ELSE
	sQuery := 'select * from t_log where severity = NULL';
END_IF
IF xFilterByDate THEN
	STU.StrConcatA(pstTo := ADR(sQuery), pstFrom := ADR(' AND timestamp < '), iBufferSize := TO_INT(XSIZEOF(sQuery)));
	SysMem.SysMemSet(pDest := ADR(sAux), udiCount := XSIZEOF(sAux), udiValue := 0);
	sAux := SysD_DB.FUN_ConvertToSQLQueryString(sString := sFilter_LastEventDT);
	STU.StrConcatA(pstTo := ADR(sQuery), pstFrom := ADR(sAux), iBufferSize := TO_INT(XSIZEOF(sQuery)));
END_IF
IF xFilterByComponent THEN
	STU.StrConcatA(pstTo := ADR(sQuery), pstFrom := ADR(' AND component = '), iBufferSize := TO_INT(XSIZEOF(sQuery)));
	SysMem.SysMemSet(pDest := ADR(sAux), udiCount := XSIZEOF(sAux), udiValue := 0);
	sAux := SysD_DB.FUN_ConvertToSQLQueryString(sString := sFilter_Component);
	STU.StrConcatA(pstTo := ADR(sQuery), pstFrom := ADR(sAux), iBufferSize := TO_INT(XSIZEOF(sQuery)));
END_IF

xContinueGetLog := xAppendToExtendedLog AND diLastNonNullLogID > 0;//02/11/2022
IF xContinueGetLog THEN //02/11/2022
	STU.StrConcatA(pstTo := ADR(sQuery), pstFrom := ADR(' AND id < '), iBufferSize := TO_INT(XSIZEOF(sQuery)));
	sAux := TO_STRING(diLastNonNullLogID);
	STU.StrConcatA(pstTo := ADR(sQuery), pstFrom := ADR(sAux), iBufferSize := TO_INT(XSIZEOF(sQuery)));
END_IF

STU.StrConcatA(pstTo := ADR(sQuery), pstFrom := ADR(' order by id desc limit 40'), iBufferSize := TO_INT(XSIZEOF(sQuery)));

diQueryLength := STU.StrLenA(pstData := ADR(sQuery));

eQueryError := SysD_DB.FUN_Query2SQLCmd(
	pbQuery := ADR(sQuery), 
	diQueryLength := diQueryLength,
	asSQLCommand => asMySQLCommand	
);

SysMem.SysMemSet(pDest := ADR(aLog), udiCount := XSIZEOF(aLog), udiValue := 0);

pInterpDest := ADR(aLog);
uiDimInterpDest := __UXINT_TO_UINT(XSIZEOF(aLog)/XSIZEOF(aLog[0]));

itfInterpreter := SQL_Interp_GetLog_0;

REF_REQ_SQLQuery REF= REQ_GetLog;

eMySQLAction := SysD_DB.SysD_DB_actions_enum_t.Query;


                      
END_ACTION

ACTION ACT_GetLog_Success:
                        IF eLastInterpError = SysD_DB.ERROR.NO_ERROR THEN
// 	diActionID := aSAPA_RequestedActions[0].diID;
	METH_CopyToExtendedLog();
ELSIF eLastInterpError = SysD_DB.ERROR.NULL_RESULT THEN
	diActionID := -1;
END_IF
                      
END_ACTION

ACTION ACT_SingleInsert:
                        // SINGLE INSERT
ePollRes := itfQueue_LogEntries.Poll(itfElement => itfElement);
xResult := __QUERYINTERFACE(itfElement, itfLogEntryElement);
IF xResult THEN
	LogEntryToInsert := itfLogEntryElement.LogEntry;
	xLogEntryIsValid := METH_LogEntryIsValid(LogEntry := LogEntryToInsert);
	IF xLogEntryIsValid THEN // single insert
		xTB_InsertLogEntry := TRUE;
	END_IF
END_IF
                      
END_ACTION

ACTION ACT_MultiInsert:
                        ePollRes := COL.COLLECTION_ERROR.NO_ERROR;
sMultiInsertQuery := '';
WHILE METH_MultiInsertCond() DO
	diMultiInsertQueryLen := STU.StrLenA(pstData := ADR(sMultiInsertQuery));
	
	ePeekRes := itfQueue_LogEntries.Peek(itfElement => itfElement);
	xResult := __QUERYINTERFACE(itfElement, itfLogEntryElement);
	IF xResult THEN
		LogEntryToInsert := itfLogEntryElement.LogEntry;
		xLogEntryIsValid := METH_LogEntryIsValid(LogEntry := LogEntryToInsert);
		IF xLogEntryIsValid THEN
			sPeekQuery := '';
			sPeekQuery := FUN_DB_insert_log_entry(
				SysD_LogEntry := LogEntryToInsert,
			);
			
			diPeekQueryLen := STU.StrLenA(pstData := ADR(sPeekQuery));
			diSumQueryLen := diMultiInsertQueryLen + diPeekQueryLen;
			diMaxQueryLen := TO_DINT(XSIZEOF(sMultiInsertQuery)) - 1;
			xAddToMultiInsert := diSumQueryLen < diMaxQueryLen;
			IF xAddToMultiInsert THEN
				// concatenate the peeked string to the query
				xConcatRes := STU.StrConcatA(
					pstTo := ADR(sMultiInsertQuery), 
					pstFrom := ADR(sPeekQuery), 
					iBufferSize := TO_INT(XSIZEOF(sMultiInsertQuery))
				);
				ePollRes := itfQueue_LogEntries.Poll(itfElement => itfElement); // poll the element
			ELSE // don't poll, leave it for the next round
				EXIT;
			END_IF
		ELSE // eliminate by polling
			eRemoveRes := itfQueue_LogEntries.Poll(itfElement => itfElement);
		END_IF
	END_IF
END_WHILE
IF sMultiInsertQuery <> '' THEN
	xTB_MultiInsertLogEntries := TRUE;
END_IF
                      
END_ACTION

METHOD METH_LogEntryIsValid : BOOL
  VAR_INPUT
    LogEntry : SysD_log_entry_t;
  END_VAR
                          METH_LogEntryIsValid := 
	LogEntry.sTimeStamp <> ''
	AND LogEntry.sDescription <> ''
;
                        
END_METHOD

METHOD METH_GetLastNonNullID : DINT
  VAR_INPUT
    pLog : POINTER TO SysD_log_row_t;
    udiDim : UDINT;
  END_VAR
  VAR_OUTPUT
    udiArrayInd : UDINT := 0;
    xEmptyArray : BOOL := TRUE;
  END_VAR
  VAR
    udiInd : UDINT;
    pCurrentLog : POINTER TO SysD_log_row_t;
    diRes : DINT := -1;
    xParsingOK : BOOL;
  END_VAR
                          xParsingOK := pLog > 0 AND udiDim > 0;
IF xParsingOK THEN
	WHILE udiInd < udiDim DO
		pCurrentLog := pLog + TO___XWORD(udiInd) * XSIZEOF(pLog^);
		IF pCurrentLog^.diID = 0 THEN
			EXIT;
		ELSE
			xEmptyArray := FALSE;
			diRes := pCurrentLog^.diID;
			udiArrayInd := udiInd;
			udiInd := udiInd + 1;
		END_IF
	END_WHILE
END_IF

METH_GetLastNonNullID := diRes;
                        
END_METHOD

METHOD METH_CopyToExtendedLog : BOOL
  VAR
    udiExtLastNonNullArrInd : UDINT;
    xExtIsEmptyArray : BOOL;
    diExtLastNonNullLogID : DINT;
    diLocalLastNonNullLogID : DINT;
    xLocalIsEmptyArray : BOOL;
    udiLocalLastNonNullArrInd : UDINT;
    udiExtInd : UDINT;  (* where to copy *)
    udiLocalInd : UDINT;  (* what to copy *)
    pCurrExt : POINTER TO SysD_log_row_t;
    pCurrLocal : POINTER TO SysD_log_row_t;
  END_VAR
                          diExtLastNonNullLogID := METH_GetLastNonNullID(
	pLog := ADR(aExtendedLog), udiDim := udiDimExtendedLog,
	udiArrayInd => udiExtLastNonNullArrInd,
	xEmptyArray => xExtIsEmptyArray
);

diLocalLastNonNullLogID := METH_GetLastNonNullID(
	pLog := ADR(aLog), udiDim := udiDimLog,
	udiArrayInd => udiLocalLastNonNullArrInd,
	xEmptyArray => xLocalIsEmptyArray
);

IF xExtIsEmptyArray THEN
	udiExtInd := 0;
ELSE
	udiExtInd := udiExtLastNonNullArrInd + 1;
END_IF
udiLocalInd := 0;
WHILE udiExtInd < udiDimExtendedLog AND udiLocalInd <= udiLocalLastNonNullArrInd DO
	pCurrExt := ADR(aExtendedLog) + udiExtInd * XSIZEOF(pCurrExt^);
	pCurrLocal := ADR(aLog) + udiLocalInd * XSIZEOF(pCurrExt^);
	pCurrExt^ := pCurrLocal^; //copy
	
	udiExtInd := udiExtInd + 1;
	udiLocalInd := udiLocalInd + 1;
END_WHILE
                        
END_METHOD

METHOD METH_AddEntryToQueue : COL.COLLECTION_ERROR
  VAR_INPUT
    LogEntry : SysD_log_entry_t;
    pdiCounter : POINTER TO DINT := 0;
  END_VAR
  VAR_OUTPUT
    xFullBuffer : BOOL;
    sLastTimestamp : STRING;
  END_VAR
  VAR
    eRes : COL.COLLECTION_ERROR;
    xAddOk : BOOL;
  END_VAR
                          LogEntry.sTimeStamp := FUN_GetLocalRTCString();
eRes := itfQueue_LogEntries.AddElement(
	itfElement := LogEntriesFactory.Create(
		Value := LogEntry, 
		eError => eLogEntryFactErr
	)
);
xAddOk := eRes = COL.COLLECTION_ERROR.NO_ERROR AND eLogEntryFactErr = FBF.ERROR.NO_ERROR;
IF xAddOk THEN
// 	diCounter := (diCounter + 1) MOD 16#7FFFFFFF;
	IF pdiCounter > 0 THEN //increment counter if passed as pointer
		pdiCounter^ := pdiCounter^ + 1;
	END_IF
	sLastTimestamp := LogEntry.sTimeStamp;
ELSE
	xFullBuffer := eRes = COL.COLLECTION_ERROR.MAXIMUM_SIZE_OF_ELEMENTS_EXCEEDED;
END_IF
                        
END_METHOD

METHOD METH_MultiInsertCond : BOOL
  VAR
    udiEntries : UDINT;
    diMaxQueryLen : DINT;
    diQueryLenThreshold : DINT;
  END_VAR
                          udiEntriesToInsert := itfQueue_LogEntries.CountElements();
diMultiInsertQueryLen := STU.StrLenA(pstData := ADR(sMultiInsertQuery));
diMaxQueryLen := TO_DINT(XSIZEOF(sQuery)) - 1;
diQueryLenThreshold := TO_DINT(TO_REAL(diMaxQueryLen) * 0.75);
// diPeekQueryLen := STU.StrLenA(pstData := ADR(sPeekQuery));

METH_MultiInsertCond :=
	ePollRes = COL.COLLECTION_ERROR.NO_ERROR
	AND udiEntriesToInsert > 0
	AND diMultiInsertQueryLen < diQueryLenThreshold;
;
                        
END_METHOD
END_PROGRAM

PROGRAM prgDBExecutor
  VAR
    eIterResult : COL.COLLECTION_ERROR;
    COL_ListIterator : COL.ListIterator;
    itfStringElement : COL.IElement;
    itfMySQLResult : SysD_DB.IMySQLResultElement;
    xResultIt : BOOL;
    iftStringKey : COL.IStringElement;
    itfElement : COL.IElement;
    xInspectHashtable : BOOL;
    MySQLResult : SysD_DB.SysD_DB_result_struct_t;
    xInspectQueue : BOOL;
    eIterRequest : COL.COLLECTION_ERROR;
    itfMySQLRequest : SysD_DB.IMySQLRequestElement;
    MySQLRequest : SysD_DB.SysD_DB_request_struct_t;
    sTestDBName : STRING := 'db_sapa_test';
    xTB_TESTDB : BOOL;
    xIsTest : BOOL;
    asIN_MySQLRequests : ARRAY[0..c_uiMaxIndArray] OF SysD_DB.IMySQLRequestElement;  (* QUEUE IN *)
    itfINQueue_MySQLRequest : COL.Queue := (paElements := ADR(asIN_MySQLRequests), udiMaxElements := UINT_TO_UDINT((c_uiMaxIndArray + 1)));
    HashTableFactory : COL.HashTableFactory;  (* Factory to create a hash table on heap memory. *)
    itfOUTHashTable_MySQLResult : COL.IMap := HashTableFactory.Create(udiMaxElements := UINT_TO_UDINT((c_uiMaxIndArray + 1)));  (* Creates a hashtable on heap memory. NOTE: Collections that have been created with this Factory are not online change safe. *)
    iCountFailure : INT;
    eLastExecutorError : SysD_DB.EXECUTOR_ERROR;
    udiINRequestsNum : UDINT;
    udiOUTResultsNum : UDINT;
    iMaxClients : INT := 2;
    SysD_DB_Executor_0 : SysD_DB.SysD_DB_Executor;
    CTRL_Executor : SysDesignBasic.SysD_basic_ctrl_struct_t := (xExecute := TRUE);
    eMySQLExecutorError : SysD_DB.EXECUTOR_ERROR;
    ClientsOccupationStatistic : SysD_DB.SysD_DB_clients_occ_stat_struct_t;
    aeClientsOccupation : ARRAY[0..SysD_DB.Constants.gc_uiMaxIndMySQLClients] OF SysD_DB.SysD_DB_client_state_enum_t;
  END_VAR
  VAR CONSTANT
    c_uiMaxIndArray : UINT := 49;
  END_VAR

                    (*--------------------------*)
// 2/12/2022: set database

(*--------------------------*)

udiINRequestsNum := itfINQueue_MySQLRequest.CountElements();
udiOUTResultsNum := itfOUTHashTable_MySQLResult.CountKeys();

SysD_DB_Executor_0(
	xEnable := CTRL_Executor.xExecute,
	xBusy => CTRL_Executor.xProcessing,
	xError => CTRL_Executor.xFailure,
	
	eErrorID => eMySQLExecutorError,
	
	pIN_Queue := ADR(itfINQueue_MySQLRequest),
	pOUT_Hashtable := ADR(itfOUTHashTable_MySQLResult),
	iMaxClients := iMaxClients,
	
	ClientsOccupationStatistic => ClientsOccupationStatistic,
	aeClientsOccupation => aeClientsOccupation
);
CTRL_Executor.xTerminated := CTRL_Executor.xFailure;
IF CTRL_Executor.xTerminated THEN
	eLastExecutorError := eMySQLExecutorError;
	IF CTRL_Executor.xSuccess THEN
		// never
	ELSIF CTRL_Executor.xFailure THEN
		iCountFailure := (iCountFailure + 1) MOD 16#7FFF;
	END_IF
	CTRL_Executor.xExecute := FALSE;
	SysD_DB_Executor_0(xEnable := FALSE);
END_IF
(*=====================================================*)
//21/12/2022: debugging
// IF xInspectHashtable THEN
// 	eIterResult := itfOUTHashTable_MySQLResult.Keys(itfIterator := COL_ListIterator);
// 	IF eIterResult = COL.COLLECTION_ERROR.NO_ERROR THEN
// 		WHILE COL_ListIterator.HasNext() DO
// 			COL_ListIterator.Next(itfElement => itfStringElement);
// 			xResultIt :=  __QUERYINTERFACE(itfStringElement, iftStringKey);
// 			IF xResultIt THEN
// 				itfOUTHashTable_MySQLResult.GetElementByKey(itfKey := iftStringKey, itfValue => itfElement);
// 				xResultIt :=  __QUERYINTERFACE(itfElement, itfMySQLResult);
// 				IF xResultIt THEN 
// 					MySQLResult := itfMySQLResult.PROP_MySQLResultElement;
// 				END_IF
// 			END_IF
// 		END_WHILE;
// 	END_IF
// END_IF
// IF xInspectQueue THEN
// 	eIterRequest := itfINQueue_MySQLRequest.ElementIterator(itfIterator := COL_ListIterator);
// 	IF eIterRequest = COL.COLLECTION_ERROR.NO_ERROR THEN
// 		WHILE COL_ListIterator.HasNext() DO
// 			COL_ListIterator.Next(itfElement => itfElement);
// 			xResultIt :=  __QUERYINTERFACE(itfElement, itfMySQLRequest);
// 			IF xResultIt THEN
// 				MySQLRequest := itfMySQLRequest.PROP_MySQLRequestElement;
// 			END_IF
// 		END_WHILE;
// 	END_IF
// END_IF

                  
END_PROGRAM

(* Implicitly generated code : DO NOT EDIT *)
{attribute 'check_pointer'}
{attribute 'no_check'}
FUNCTION CheckPointer : POINTER TO BYTE
  VAR_INPUT
    ptToTest : POINTER TO BYTE;  (* Destination address of the pointer *)
    iSize : DINT;  (* Size of the type the pointer points to. (e.g: 20 for POINTER TO ARRAY [0..9] OF INT) *)
    iGran : DINT;  (* Granularity of the pointer access. This is the size of the biggest non-structured data type in the type the pointer points to. (e.g: 2 for POINTER TO ARRAY [0..9] OF INT) *)
    bWrite : BOOL;  (* Indicates read or write access. TRUE = write access. *)
  END_VAR
  VAR
    xError : BOOL;
  END_VAR

                    // No standard way of implementation. Fill your own code here.
IF ptToTest = 0 THEN
	xError := TRUE;
END_IF
CheckPointer := ptToTest;
                  
END_FUNCTION

PROGRAM prgInboundSync
  VAR
    BoxAtGateInfo : INCAS_box_info_struct_t;
    xNewBox : BOOL;
    sBoxInfoFromDB : db_t_items_struct_t;
    xInfoReceived : BOOL;
    xDelayBoxInMachineCond : BOOL;
    TON_DelayBoxInMachine : TON;
    tDelay : TIME := TIME#5s0ms;
    BoxAckFeedback : INCAS_box_ack_struct_t;
    iResSetFeedback : INT;
    iAnalyzeRes : INT;
    eErrorID : INCAS_box_error_enum_t;
  END_VAR

                    (*-----------------------------------------*)
// New box on OPC UA
IF xNewBox THEN
	xNewBox := FALSE;
	prgDBQuerier_SorterSX.METH_GetBoxInfo(sBoxCode := BoxAtGateInfo.box_code);
	SysMemSet(pDest := ADR(BoxAckFeedback), udiCount := XSIZEOF(BoxAckFeedback), udiValue := 0);
	BoxAckFeedback.last_box_code := BoxAtGateInfo.box_code;
	BoxAckFeedback.time_stamp := FUN_GetLocalRTCString();
	BoxAckFeedback.error_id := TO_INT(INCAS_box_error_enum_t.BUSY);
	iResSetFeedback := prgOPCUAIncas.METH_SetIncasInboundFeedback_01(
		Feedback := BoxAckFeedback
	);
END_IF
(*-----------------------------------------*)
// info received from DB
IF xInfoReceived THEN
	xInfoReceived := FALSE;
	iAnalyzeRes := METH_AnalyzeBoxInfo(
		InfoOnOPCUa := BoxAtGateInfo,
		InfoOnDb := sBoxInfoFromDB,
		eErrorID => eErrorID
	);
	xDelayBoxInMachineCond := TRUE;
	BoxAckFeedback.time_stamp := FUN_GetLocalRTCString();
	BoxAckFeedback.error_id := TO_INT(eErrorID);
	iResSetFeedback := prgOPCUAIncas.METH_SetIncasInboundFeedback_01(
		Feedback := BoxAckFeedback
	);
END_IF
(*-----------------------------------------*)
// take over
TON_DelayBoxInMachine(IN := xDelayBoxInMachineCond, PT := tDelay);
IF TON_DelayBoxInMachine.Q THEN
	xDelayBoxInMachineCond := FALSE;
	BoxAckFeedback.time_stamp := FUN_GetLocalRTCString();
	BoxAckFeedback.error_id := TO_INT(INCAS_box_error_enum_t.BOX_TAKEN_OVER);
	prgOPCUAIncas.METH_SetIncasInboundFeedback_01(
		Feedback := BoxAckFeedback
	);
END_IF
                  

METHOD METH_NewBoxAtGate : INT
  VAR_INPUT
    BoxInfo : INCAS_box_info_struct_t;
  END_VAR
  VAR
    iRes : INT;
  END_VAR
                          IF BoxInfo.box_code <> '' THEN
	BoxAtGateInfo := BoxInfo;
	xNewBox := TRUE;
ELSE
	iRes := -1;
END_IF
METH_NewBoxAtGate := iRes;
                        
END_METHOD

METHOD METH_NotifyBoxInfo : INT
  VAR_INPUT
    ItemInfo : db_t_items_struct_t;
  END_VAR
                          sBoxInfoFromDB := ItemInfo;
xInfoReceived := TRUE;
                        
END_METHOD

METHOD METH_AnalyzeBoxInfo : INT
  VAR_INPUT
    InfoOnOPCUa : INCAS_box_info_struct_t;
    InfoOnDb : db_t_items_struct_t;
  END_VAR
  VAR_OUTPUT
    eErrorID : INCAS_box_error_enum_t;
  END_VAR
  VAR
    xBoxNotFound : BOOL;
    xDimInfoMatching : BOOL;
    xToDiscard : BOOL;
    xSameBox : BOOL;
    xOk : BOOL;
    xInfoMatching : BOOL;
  END_VAR
                          
xBoxNotFound := InfoOnDb.sBoxCode = '';
xSameBox := InfoOnOPCUa.box_code = InfoOnDb.sBoxCode;
xDimInfoMatching := InfoOnOPCUa.dim_code = InfoOnDb.sDimCode;
xInfoMatching := xDimInfoMatching;
xToDiscard := 
	InfoOnOPCUa.box_state = TO_INT(INCAS_box_state_enum_t.BOX_STATE_TO_DISCARD)
;
xOk := 
	NOT xBoxNotFound
	AND xInfoMatching
	AND xSameBox
	AND InfoOnOPCUa.box_state = TO_INT(INCAS_box_state_enum_t.BOX_STATE_AT_GATE)
;

IF xBoxNotFound THEN
	eErrorID := INCAS_box_error_enum_t.BOX_NOT_FOUND;
ELSIF NOT xInfoMatching THEN
	eErrorID := INCAS_box_error_enum_t.INFO_NOT_MATCHING;
ELSIF xToDiscard THEN
	eErrorID := INCAS_box_error_enum_t.TO_DISCARD;
ELSIF xOk THEN
	eErrorID := INCAS_box_error_enum_t.BOX_ACCEPTED;
ELSE
	eErrorID := INCAS_box_error_enum_t.TO_DISCARD;
END_IF
                        
END_METHOD
END_PROGRAM

FUNCTION FUN_GetLocalRTCString : STRING
  VAR
    dwRTC : DWORD;
    RTS_RTCRes : SysTypes.RTS_IEC_RESULT;
    dtRTCTime : DT;
    sRTCTime : STRING;
    udiResUTCLocal : SysTypes.RTS_IEC_RESULT;
    dwRTC_Local : DWORD;
    udiHighRes : SysTypes.RTS_IEC_RESULT;
    uliHighResTimestamp : SYSTIME;
    dwMilliSec : DWORD;
    sAux : STRING(255);
  END_VAR

                    udiHighRes := SysTimeRtc.SysTimeRtcHighResGet(pTimestamp := uliHighResTimestamp);
dwMilliSec := TO_DWORD(uliHighResTimestamp MOD 1000);//02/11/2022
sAux := TO_STRING(dwMilliSec);
IF dwMilliSec < 10 THEN
	sAux := CONCAT('00', sAux);
ELSIF dwMilliSec < 100 THEN
	sAux := CONCAT('0', sAux);
END_IF
dwRTC := TO_DWORD(uliHighResTimestamp / 1000);
udiResUTCLocal := SysTimeRTCConvertUTCToLocal(dwTimestampUtc := dwRTC, pdwTimestampLocal := dwRTC_Local);
dtRTCTime := DWORD_TO_DT(dwRTC_Local);
sRTCTime := DT_TO_STRING(dtRTCTime);
sRTCTime := CONCAT(sRTCTime, '.');
sRTCTime := CONCAT(sRTCTime, sAux);

FUN_GetLocalRTCString := sRTCTime;
                  
END_FUNCTION

PROGRAM prg_Hmi_OPCUATests
  VAR
    xDIS_TESTIsATest : BOOL;
    sDescriptionBar : STRING(255) := 'Stato applicazione:';
    sStatusMessage : STRING(255);
  END_VAR

                    xDIS_TESTIsATest := FALSE;
                  
END_PROGRAM

PROGRAM prg_Hmi_RobotSelection
  VAR
    sDescriptionBar : STRING(255) := 'Stato applicazione:';
    sStatusMessage : STRING(255);
  END_VAR

                    
                  

METHOD METH_IsGazelle : BOOL
                          METH_IsGazelle := prgMain.sHostName = 'gazelle';
                        
END_METHOD
END_PROGRAM

PROGRAM prgDial_ROSInfo_A
  VAR
    xIsRunning : BOOL;
    eProcessState : process_code_enum_t;
    diProcessCode : DINT;
  END_VAR

                    xIsRunning := prgROS.ROSInterface_01.ROS2Codesys.Subscripted.is_running;
eProcessState := prgROS.ROSInterface_01.ROS2Codesys.eProcessState;
diProcessCode := prgROS.ROSInterface_01.ROS2Codesys.Subscripted.process_code;
                  
END_PROGRAM

PROGRAM prgDial_ROSInfo_B
  VAR
    xIsRunning : BOOL;
    eProcessState : process_code_enum_t;
    diProcessCode : DINT;
  END_VAR

                    xIsRunning := prgROS.ROSInterface_02.ROS2Codesys.Subscripted.is_running;
eProcessState := prgROS.ROSInterface_02.ROS2Codesys.eProcessState;
diProcessCode := prgROS.ROSInterface_02.ROS2Codesys.Subscripted.process_code;
                  
END_PROGRAM

PROGRAM prg_hmi_Synoptic

                    
                  
END_PROGRAM

PROGRAM prg_hmi_Sorter_SX
  VAR
    xTB_TESTConvert : BOOL;
    TESTItem : items_struct_t := (eLocationType := location_type_enum_t.Buffer, iLocationIndex := 2, iLocationSubIndex := 1, sItemCode := 'TESTConvertBox');
    eConvertError : SORTER_MAPPING_ERROR_ENUM_T;
    xInit : BOOL := TRUE;
    sTESTConvertedLocationName : STRING;
    xEnableDrawConvertedBox : BOOL := TRUE;
    aBuffers : ARRAY[0..GVL_Consts.gc_iMaxIndBuffers] OF buffer_struct_t;  (* input substructures are externally updated, output substructures directly set IOs *)
    Conveyor : conveyor_struct_t;
    aTESTBuffers : ARRAY[0..GVL_Consts.gc_iMaxIndBuffers] OF buffer_struct_t;  (* input substructures are externally updated, output substructures directly set IOs *)
    TESTConveyor : conveyor_struct_t;
    xTEST : BOOL := TRUE;
    iBufferVisibleNum : INT;
    iConveyorVisibleNum : INT;
    sTESTLocationName : STRING := 'SorterSX-B-BufferFront1';
    xTB_TESTDraw : BOOL;
    TESTMappingInfo : mapping_info_struct_t;
    eMapError : sorter_mapping_error_enum_t;
    eDrawError : sorter_mapping_error_enum_t;
    pTESTBoxInfo : POINTER TO synoptic_boxes_info_struct_t;
    xEnableDraw : BOOL := TRUE;
    iBoxCodeRes : INT;
    sTESTBoxCode : STRING := 'TEST BOX';
    xCanWrite : BOOL;
    xTB_Clear : BOOL;
    aaBoxesBuffer : ARRAY[0..GVL_Consts.gc_iMaxIndBuffers] OF ARRAY[0..GVL_Consts.gc_uiMaxIndBuffer] OF synoptic_boxes_info_struct_t;
    aaBoxesConveyor : ARRAY[0..GVL_Consts.gc_uiMaxIndConveyor] OF synoptic_boxes_info_struct_t;
    aaTMPBoxesBuffer : ARRAY[0..GVL_Consts.gc_iMaxIndBuffers] OF ARRAY[0..GVL_Consts.gc_uiMaxIndBuffer] OF synoptic_boxes_info_struct_t;
    aaTMPBoxesConveyor : ARRAY[0..GVL_Consts.gc_uiMaxIndConveyor] OF synoptic_boxes_info_struct_t;
  END_VAR
  VAR CONSTANT
    c_iGateConveyorIndex : INT := 0;  (* conveyor *)
    c_iExitConveyorIndex : INT := 8;
    c_sSorterName : STRING := 'SorterSX';
    c_sFirstSectionName : STRING := 'B';  (* sections *)
    c_sSecondSectionName : STRING := 'F';
    c_iFirstPosIndInSecondSection : INT := 4;
    c_iLastPosIndInSecondSection : INT := 7;
    c_iMaxIndDepthBuffer : INT := 2;
    c_sDepthInterchange : STRING := 'Front';  (* buffer depth *)
    c_sDepthInternal : STRING := 'F';
    c_sDepthExternal : STRING := 'R';
  END_VAR

                    IF xInit THEN
	xInit := FALSE;
	METH_SetTESTPhysicalMapping();
END_IF

IF xTEST THEN
	aBuffers := aTESTBuffers;
	Conveyor := TESTConveyor;
END_IF

IF xTB_Clear THEN
	xTB_Clear := FALSE;
	SysMem.SysMemSet(pDest := ADR(aaTMPBoxesBuffer), udiCount := XSIZEOF(aaTMPBoxesBuffer), udiValue := 0);
	SysMem.SysMemSet(pDest := ADR(aaTMPBoxesConveyor), udiCount := XSIZEOF(aaTMPBoxesConveyor), udiValue := 0);
	aaBoxesBuffer := aaTMPBoxesBuffer;
	aaBoxesConveyor := aaTMPBoxesConveyor;
END_IF

IF xTB_TESTDraw THEN
	xTB_TESTDraw := FALSE;
	
	SysMem.SysMemSet(pDest := ADR(aaTMPBoxesBuffer), udiCount := XSIZEOF(aaTMPBoxesBuffer), udiValue := 0);
	SysMem.SysMemSet(pDest := ADR(aaTMPBoxesConveyor), udiCount := XSIZEOF(aaTMPBoxesConveyor), udiValue := 0);
	
	eDrawError := METH_Draw(
		sLocationName := sTESTLocationName,
		sBoxCode := sTESTBoxCode,
		MappingInfo => TESTMappingInfo
	);
	
	aaBoxesBuffer := aaTMPBoxesBuffer;
	aaBoxesConveyor := aaTMPBoxesConveyor;	
END_IF

IF xTB_TESTConvert THEN
	xTB_TESTConvert := FALSE;
	eConvertError := METH_ConvertItemInfoToLocationName(
		aBuffers := aTESTBuffers,
		Conveyor := TESTConveyor,
		Item := TESTItem,
		sLocationName => sTESTConvertedLocationName
	);
	
	IF xEnableDrawConvertedBox THEN
		METH_TESTDrawBox(
			sLocationName :=  sTESTConvertedLocationName,
			sBoxCode := TESTItem.sItemCode
		);
	END_IF
END_IF

(*================================================*)
iBufferVisibleNum := METH_BufferVisibility();
iConveyorVisibleNum := METH_ConveyorVisibility();



                  

METHOD METH_BufferVisibility : INT
  VAR
    iMaxIndBuffer : INT;
    iMaxIndDepth : INT;
    iIndBuffer : INT;
    iIndDepth : INT;
    xShowCond : BOOL;
    iRes : INT;
  END_VAR
                          iMaxIndBuffer := TO_INT(XSIZEOF(aaBoxesBuffer)/XSIZEOF(aaBoxesBuffer[0])) - 1;
iMaxIndDepth := TO_INT(XSIZEOF(aaBoxesBuffer[0])/XSIZEOF(aaBoxesBuffer[0][0])) - 1;

FOR iIndBuffer := 0 TO iMaxIndBuffer DO
	FOR iIndDepth := 0 TO iMaxIndDepth DO
		xShowCond := aaBoxesBuffer[iIndBuffer][iIndDepth].sBoxCode <> '';
		aaBoxesBuffer[iIndBuffer][iIndDepth].xInvisible := NOT xShowCond;
		IF xShowCond THEN
			iRes := iRes + 1;
		END_IF
	END_FOR
END_FOR

METH_BufferVisibility := iRes;
                        
END_METHOD

METHOD METH_ConveyorVisibility : INT
  VAR
    iMaxInd : INT;
    iInd : INT;
    xShowCond : BOOL;
    iRes : INT;
  END_VAR
                          iMaxInd := TO_INT(XSIZEOF(aaBoxesBuffer)/XSIZEOF(aaBoxesBuffer[0])) - 1;

FOR iInd := 0 TO iMaxInd DO
	xShowCond := aaBoxesConveyor[iInd].sBoxCode <> '';
	aaBoxesConveyor[iInd].xInvisible := NOT xShowCond;
	IF xShowCond THEN
		iRes := iRes + 1;
	END_IF
END_FOR

METH_ConveyorVisibility := iRes;
                        
END_METHOD

METHOD METH_Map : sorter_mapping_error_enum_t
  VAR_INPUT
    sLocationName : STRING;
  END_VAR
  VAR_OUTPUT
    MappingInfo : mapping_info_struct_t;
  END_VAR
  VAR
    eRes : sorter_mapping_error_enum_t;
    xIsBuffer : BOOL;
    xIsConveyor : BOOL;
    iBufferKeyFound : INT;
    aiConveyorKeyFound : ARRAY[0..c_iMaxIndConv] OF INT;
    iIndConv : INT;
    iMaxIndConv : INT;
    iBufferFrontKeyFound : INT;
    xIsBackSection : BOOL;
    xIsFrontSection : BOOL;
    xValidSection : BOOL;
    iBufferNum : INT;
    xValidBufferNum : BOOL;
    iBufferDepth : INT;
    xValidBufferDepth : BOOL;
    xParsingOK : BOOL;
    xIsGate : BOOL;
    xIsRoller : BOOL;
    sBackSectionKey : STRING;
    sFrontSectionKey : STRING;
  END_VAR
  VAR CONSTANT
    c_iMaxIndConv : INT := 2;
    c_sBufferTypeKey : STRING := 'BUFFER';
    c_asConveyorTypeKey : ARRAY[0..c_iMaxIndConv] OF STRING := ['GATE', 'ROLLER'];
    c_sBufferFrontKey : STRING := 'Front';
  END_VAR
                          xParsingOK := sLocationName <> '';
IF xParsingOK THEN // check if BUFFER
	MappingInfo.sLocationName := sLocationName;
	
	iBufferKeyFound := STU.StrCaseFindA(
		pst1 := ADR(sLocationName), 
		pst2 := ADR(c_sBufferTypeKey), 
		uiSearchStart := 0 
	);
	xIsBuffer := iBufferKeyFound > 0;
	IF xIsBuffer THEN
		MappingInfo.eType := sorter_elem_type_enum_t.Buffer;
		
		// identify which sorter section
		sBackSectionKey := CONCAT('-', CONCAT(c_sFirstSectionName, '-'));
		sFrontSectionKey := CONCAT('-', CONCAT(c_sSecondSectionName, '-'));
		xIsBackSection := FIND(sLocationName, sBackSectionKey) > 0;
		xIsFrontSection := FIND(sLocationName, sFrontSectionKey) > 0;
		xValidSection := xIsBackSection OR xIsFrontSection;
		
		IF xValidSection THEN
			IF xIsFrontSection THEN
				MappingInfo.Info.BufferInfo.iSectionIndex := 1;
			ELSE
				MappingInfo.Info.BufferInfo.iSectionIndex := 0;
			END_IF
			
			// identify buffer number
			iBufferNum := METH_FindBufferNum(
				sLocationName := sLocationName
			);
			xValidBufferNum := iBufferNum > 0;
			IF xValidBufferNum THEN
				MappingInfo.Info.BufferInfo.iNumber := iBufferNum;
				
				// identify buffer depth
				iBufferDepth := METH_FindBufferDepth(
					sLocationName := sLocationName
				);
				xValidBufferDepth := iBufferDepth >= 0;
				IF xValidBufferDepth THEN
					 MappingInfo.Info.BufferInfo.iDepth := iBufferDepth;
				ELSE
					eRes := sorter_mapping_error_enum_t.INVALID_BUFFER_DEPTH;
				END_IF
			ELSE
				eRes := sorter_mapping_error_enum_t.INVALID_BUFFER_NUMBER;
			END_IF
		ELSE
			eRes := sorter_mapping_error_enum_t.INVALID_BUFFER_SECTION;
		END_IF
	ELSE // check if CONVEYOR
		iMaxIndConv := c_iMaxIndConv;
		xIsConveyor := FALSE;
		FOR iIndConv := 0 TO iMaxIndConv DO
			aiConveyorKeyFound[iIndConv] := STU.StrCaseFindA(
				pst1 := ADR(sLocationName), 
				pst2 := ADR(c_asConveyorTypeKey[iIndConv]), 
				uiSearchStart := 0 
			);
			xIsConveyor := xIsConveyor OR (aiConveyorKeyFound[iIndConv] > 0);
			IF xIsConveyor THEN
				EXIT;
			END_IF
		END_FOR
		IF xIsConveyor THEN
			MappingInfo.eType := sorter_elem_type_enum_t.Conveyor;
			xIsGate := STU.StrCaseFindA(
				pst1 := ADR(sLocationName), 
				pst2 := ADR(c_asConveyorTypeKey[0]), 
				uiSearchStart := 0 
			) > 0;
			IF xIsGate THEN
				MappingInfo.Info.ConveyorInfo.iLocationIndex := c_iGateConveyorIndex;
			ELSE
				xIsRoller := STU.StrCaseFindA(
					pst1 := ADR(sLocationName), 
					pst2 := ADR(c_asConveyorTypeKey[1]), 
					uiSearchStart := 0 
				) > 0;
				IF xIsRoller THEN
					MappingInfo.Info.ConveyorInfo.iLocationIndex := c_iExitConveyorIndex;
				ELSE
					eRes := sorter_mapping_error_enum_t.INVALID_LOCATION_NAME;
				END_IF
			END_IF
		ELSE
			eRes := sorter_mapping_error_enum_t.INVALID_LOCATION_NAME;
		END_IF
	END_IF
ELSE
	eRes := sorter_mapping_error_enum_t.INVALID_INPUT;
END_IF

METH_Map := eRes;
                        
END_METHOD

METHOD METH_FindBufferNum : INT
  VAR_INPUT
    sLocationName : STRING;
  END_VAR
  VAR
    iIndNum : INT;
    iMaxIndNum : INT;
    sAux : STRING;
    xNumFound : BOOL;
    iNum : INT;
    iRes : INT := -1;
  END_VAR
                          iMaxIndNum := TO_INT(XSIZEOF(aBuffers)/XSIZEOF(aBuffers[0])) - 1;
FOR iIndNum := iMaxIndNum TO 0 BY -1 DO
	iNum := iIndNum + 1;
	sAux := TO_STRING(iNum);
	xNumFound := FIND(sLocationName, sAux) > 0;
	IF xNumFound THEN
		iRes := iNum;
		EXIT;
	END_IF
END_FOR

METH_FindBufferNum := iRes;
                        
END_METHOD

METHOD METH_FindBufferDepth : INT
  VAR_INPUT
    sLocationName : STRING;
  END_VAR
  VAR
    iRes : INT := -1;
    xIsR : BOOL;
    xIsF : BOOL;
    xIsFront : BOOL;
  END_VAR
                          xIsR := RIGHT(sLocationName, 1) = c_sDepthExternal;
xIsF := RIGHT(sLocationName, 1) = c_sDepthInternal;
xIsFront := LEFT(RIGHT(sLocationName, 6), 5) = c_sDepthInterchange;

IF xIsFront THEN
	iRes := 0;
ELSIF xIsF THEN
	iRes := 1;
ELSIF xIsR THEN
	iRes := 2;
END_IF

METH_FindBufferDepth := iRes;
                        
END_METHOD

METHOD METH_GetDrawingPointer : sorter_mapping_error_enum_t
  VAR_INPUT
    MappingInfo : mapping_info_struct_t;
    xUseTMPStructs : BOOL := TRUE;
  END_VAR
  VAR_OUTPUT
    pBoxInfo : POINTER TO synoptic_boxes_info_struct_t;
  END_VAR
  VAR
    eRes : SORTER_MAPPING_ERROR_ENUM_T;
    iStartingIndex : INT := -1;
    iOffsetIndex : INT;
    iBufferIndex : INT;
    iMaxBufferIndex : INT;
    xValidDepth : BOOL;
    iMaxDepthIndex : INT;
    iBufferDepth : INT;
    iMaxConvIndex : INT;
    xValidCondIndex : BOOL;
    iConveyorIndex : INT;
  END_VAR
                          
CASE MappingInfo.eType OF
	sorter_elem_type_enum_t.Buffer:
		CASE MappingInfo.Info.BufferInfo.iSectionIndex OF
			0:
				iStartingIndex := 0;
			1:
				iStartingIndex := 4;
			
		END_CASE
		IF iStartingIndex >= 0 THEN // valid section
			IF MappingInfo.Info.BufferInfo.iNumber > 0 THEN
				iOffsetIndex := (MappingInfo.Info.BufferInfo.iNumber - 1);
				iBufferIndex := iStartingIndex + iOffsetIndex;
				iMaxBufferIndex := TO_INT(XSIZEOF(aBuffers)/XSIZEOF(aBuffers[0])) - 1;
				IF iBufferIndex <= iMaxBufferIndex THEN // valid buffer index
					iMaxDepthIndex := TO_INT(XSIZEOF(aBuffers[0].axPositionSensors)/XSIZEOF(aBuffers[0].axPositionSensors[0])) - 1;
					iBufferDepth := MappingInfo.Info.BufferInfo.iDepth;
					xValidDepth := 
						iBufferDepth >= 0 
						AND iBufferDepth <= iMaxDepthIndex
					; 
					IF xValidDepth THEN // valid bbuffer depth
						IF xUseTMPStructs THEN
							pBoxInfo := ADR(aaTMPBoxesBuffer[iBufferIndex][iBufferDepth]);
						ELSE
							pBoxInfo := ADR(aaBoxesBuffer[iBufferIndex][iBufferDepth]);
						END_IF
					ELSE
						eRes := sorter_mapping_error_enum_t.INVALID_BUFFER_PARAMS;	
					END_IF
				ELSE
					eRes := sorter_mapping_error_enum_t.INVALID_BUFFER_PARAMS;	
				END_IF
			ELSE
				eRes := sorter_mapping_error_enum_t.INVALID_BUFFER_PARAMS;	
			END_IF
		ELSE
			eRes := sorter_mapping_error_enum_t.INVALID_BUFFER_PARAMS;			
		END_IF
	(*--------------------------------------------*)
	sorter_elem_type_enum_t.Conveyor:
		iMaxConvIndex := TO_INT(XSIZEOF(Conveyor.aLocations)/XSIZEOF(Conveyor.aLocations[0])) - 1;
		iConveyorIndex := MappingInfo.Info.ConveyorInfo.iLocationIndex;
		xValidCondIndex := 
			iConveyorIndex >= 0 
			AND iConveyorIndex <= iMaxConvIndex
		;
		IF xValidCondIndex THEN
			IF xUseTMPStructs THEN
				pBoxInfo := ADR(aaTMPBoxesConveyor[iConveyorIndex]);
			ELSE
				pBoxInfo := ADR(aaBoxesConveyor[iConveyorIndex]);
			END_IF
		ELSE
			eRes := sorter_mapping_error_enum_t.INVALID_CONVEYOR_PARAMS;	
		END_IF
	(*--------------------------------------------*)
	ELSE
		eRes := sorter_mapping_error_enum_t.INVALID_INPUT;
END_CASE
METH_GetDrawingPointer := eRes;
                        
END_METHOD

METHOD METH_WriteBoxCode : INT
  VAR_INPUT
    sBoxCode : STRING;
  END_VAR
  VAR_IN_OUT
    BoxInfo : synoptic_boxes_info_struct_t;
  END_VAR
                          BoxInfo.sBoxCode := sBoxCode;
                        
END_METHOD

METHOD METH_Draw : sorter_mapping_error_enum_t
  VAR_INPUT
    sLocationName : STRING;
    sBoxCode : STRING;
    xEnableDrawing : BOOL := TRUE;
  END_VAR
  VAR_OUTPUT
    MappingInfo : mapping_info_struct_t;
  END_VAR
  VAR
    eRes : sorter_mapping_error_enum_t;
    pBoxInfo : POINTER TO synoptic_boxes_info_struct_t;
    eDrawingError : sorter_mapping_error_enum_t;
  END_VAR
                          eMapError := METH_Map(
	sLocationName := sLocationName,
	MappingInfo => MappingInfo
);
IF eMapError = sorter_mapping_error_enum_t.NO_ERROR THEN
	eDrawingError := METH_GetDrawingPointer(
		MappingInfo := MappingInfo,
		pBoxInfo => pBoxInfo
	);
	xCanWrite := 
		eDrawingError = sorter_mapping_error_enum_t.NO_ERROR
		AND pBoxInfo > 0
	;
	IF xCanWrite THEN
		IF xEnableDraw THEN
			iBoxCodeRes := METH_WriteBoxCode(
				sBoxCode := sBoxCode,
				BoxInfo := pBoxInfo^
			);
		END_IF
	ELSE
		IF eDrawingError = sorter_mapping_error_enum_t.NO_ERROR THEN
			eRes := sorter_mapping_error_enum_t.IMPOSSIBLE_TO_DRAW;
		ELSE
			eRes := eDrawingError;
		END_IF
	END_IF
ELSE
	eRes := eMapError;
END_IF

METH_Draw := eRes;
                        
END_METHOD

METHOD METH_TESTDrawBox : INT
  VAR_INPUT
    sLocationName : STRING;
    sBoxCode : STRING := '';
  END_VAR
                          xTB_TESTDraw := TRUE;
sTESTLocationName := sLocationName;
IF sBoxCode <> '' THEN
	sTESTBoxCode := sBoxCode;
END_IF
                        
END_METHOD

METHOD METH_ConvertItemInfoToLocationName : SORTER_MAPPING_ERROR_ENUM_T
  VAR_INPUT
    aBuffers : ARRAY[0..GVL_Consts.gc_iMaxIndBuffers] OF buffer_struct_t;  (* input substructures are externally updated, output substructures directly set IOs *)
    Conveyor : conveyor_struct_t;
    Item : items_struct_t;
  END_VAR
  VAR_OUTPUT
    sLocationName : STRING;
  END_VAR
  VAR
    xValidItem : BOOL;
    eRes : SORTER_MAPPING_ERROR_ENUM_T;
    sSorterName : STRING;
    sSectionName : STRING;
    sBufferNumberName : STRING;
    sBufferLocationName : STRING;  (* sBufferDepthName : STRING; *)
    iNum : INT;
    xValidDepth : BOOL;
    sResult : STRING;
    xValidConveyorIndex : BOOL;
    sSide : STRING(2);
    iInterchageBufferIndex : INT;
    xValidSide : BOOL;
  END_VAR
                          xValidItem := METH_IsValidItem(Item := Item);
sSorterName := c_sSorterName;

IF xValidItem THEN
	CASE Item.eLocationType OF
		location_type_enum_t.Buffer:
			sSectionName := METH_GetSectionName(iIndex := Item.iLocationIndex);
			IF sSectionName <> '' THEN				
				sBufferNumberName := METH_GetBufferNumName(
					sSectionName := sSectionName, 
					iIndex := Item.iLocationIndex
				);
				
				xValidDepth := Item.iLocationSubIndex >= 0 AND Item.iLocationSubIndex <= c_iMaxIndDepthBuffer;
				IF xValidDepth THEN
					sBufferLocationName := METH_GetBufferLocationName(
						sBufferNumName := sBufferNumberName,
						iSubIndex := Item.iLocationSubIndex
					);
					
					// Compose
					sResult := METH_ComposeBufferLocationName(
						sSorterName := sSorterName,
						sSectionName := sSectionName,
						sBufferLocationName := sBufferLocationName
					);
				ELSE
					eRes := sorter_mapping_error_enum_t.ITEM_BUFFER_DEPTH_OUT_OF_BOUNDS;
				END_IF
			ELSE
				eRes := sorter_mapping_error_enum_t.ITEM_BUFFER_NUM_OUT_OF_BOUNDS;
			END_IF
		(*---------------------------------------------*)
		location_type_enum_t.Conveyor:
			xValidConveyorIndex :=
				Item.iLocationIndex >= 0 
				AND Item.iLocationIndex <= c_iExitConveyorIndex
			;
			IF xValidConveyorIndex THEN
				sSide := RIGHT(c_sSorterName, 2);
				IF Item.iLocationIndex = 0 THEN // GATE
					sResult := CONCAT('Gate-', sSide);
				ELSIF Item.iLocationIndex = c_iExitConveyorIndex THEN // EXIT ROLLER
					IF xValidSide := METH_IsValidSorterSide(sSide := sSide) THEN
						sResult := METH_GetExitLocationName(sSide := sSide);
					ELSE
						eRes := sorter_mapping_error_enum_t.INVALID_SORTER_SIDE;
					END_IF
				ELSE
					//associate with BufferFrontX corresponding position
					iInterchageBufferIndex := Conveyor.aLocations[Item.iLocationIndex].iBufferIndex;
					IF iInterchageBufferIndex >= 0 AND iInterchageBufferIndex < c_iLastPosIndInSecondSection THEN
						sSectionName := METH_GetSectionName(iIndex := iInterchageBufferIndex);
						sBufferNumberName := METH_GetBufferNumName(
							sSectionName := sSectionName, 
							iIndex := iInterchageBufferIndex
						);
						sBufferLocationName := CONCAT(c_sDepthInterchange, sBufferNumberName);
						sResult := METH_ComposeBufferLocationName(
							sSorterName := sSorterName,
							sSectionName := sSectionName,
							sBufferLocationName := sBufferLocationName
						);
					ELSE
						eRes := sorter_mapping_error_enum_t.INVALID_INTERCHANGE_LOCATION;
					END_IF
					
					
				END_IF
			ELSE
				eRes := sorter_mapping_error_enum_t.ITEM_CONVEYOR_OUT_OF_BOUNDS;
			END_IF
		(*---------------------------------------------*)
	END_CASE
ELSE
	eRes := sorter_mapping_error_enum_t.INVALID_ITEM;
END_IF

IF eRes = sorter_mapping_error_enum_t.NO_ERROR THEN
	sLocationName := sResult;
END_IF

METH_ConvertItemInfoToLocationName := eRes;
                        
END_METHOD

METHOD METH_IsValidItem : BOOL
  VAR_INPUT
    Item : items_struct_t;
  END_VAR
                          METH_IsValidItem := 
	Item.eLocationType <> location_type_enum_t.Undefined
	AND Item.sItemCode <> ''
	AND Item.iLocationIndex >= 0
	AND (Item.iLocationSubIndex >= 0 OR Item.eLocationType = location_type_enum_t.Conveyor)
;
                        
END_METHOD

METHOD METH_ComposeBufferLocationName : STRING
  VAR_INPUT
    sSorterName : STRING;
    sSectionName : STRING;
    sBufferLocationName : STRING;
  END_VAR
                          METH_ComposeBufferLocationName := CONCAT(
	sSorterName,
	CONCAT(
		'-',
		CONCAT(
			sSectionName,
			CONCAT(
				'-',
				CONCAT(
					'Buffer',
					sBufferLocationName
				)
			)
		)
	)
);
                        
END_METHOD

METHOD METH_GetSectionName : STRING
  VAR_INPUT
    iIndex : INT;
  END_VAR
  VAR
    sRes : STRING;
  END_VAR
                          IF iIndex >= 0 AND iIndex < c_iFirstPosIndInSecondSection THEN
	sRes := c_sFirstSectionName;
ELSIF iIndex >= c_iFirstPosIndInSecondSection AND iIndex < c_iLastPosIndInSecondSection THEN
	sRes := c_sSecondSectionName;
END_IF

METH_GetSectionName := sRes;
                        
END_METHOD

METHOD METH_GetBufferNumName : STRING
  VAR_INPUT
    sSectionName : STRING;
    iIndex : INT;
  END_VAR
  VAR
    iNum : INT;
    sRes : STRING;
  END_VAR
                          IF sSectionName = c_sFirstSectionName THEN
	iNum := iIndex + 1;
	sRes := TO_STRING(iNum);
ELSIF sSectionName = c_sSecondSectionName THEN
	iNum := (iIndex - c_iFirstPosIndInSecondSection) + 1;
	sRes := TO_STRING(iNum);
END_IF

METH_GetBufferNumName := sRes;
                        
END_METHOD

METHOD METH_GetBufferLocationName : STRING
  VAR_INPUT
    sBufferNumName : STRING;
    iSubIndex : INT;
  END_VAR
  VAR
    sRes : STRING;
    sBufferDepthName : STRING;
  END_VAR
                          CASE iSubIndex OF
	0:
		sBufferDepthName := c_sDepthInterchange;
		sRes := CONCAT(sBufferDepthName, sBufferNumName);
	1:
		sBufferDepthName := c_sDepthInternal;
		sRes := CONCAT(sBufferNumName, sBufferDepthName);
	2:
		sBufferDepthName := c_sDepthExternal;
		sRes := CONCAT(sBufferNumName, sBufferDepthName);
END_CASE
METH_GetBufferLocationName := sRes;
                        
END_METHOD

METHOD METH_GetExitLocationName : STRING
  VAR_INPUT
    sSide : STRING;
  END_VAR
  VAR
    sRes : STRING;
  END_VAR
                          IF sSide = 'DX' THEN
	sRes := CONCAT(
		'Roller', 
		CONCAT(
			sSide,
			'-A'
		)
	);
ELSIF sSide = 'SX' THEN
	sRes := CONCAT('Roller', RIGHT(c_sSorterName, 2));
END_IF

METH_GetExitLocationName := sRes;
                        
END_METHOD

METHOD METH_IsValidSorterSide : BOOL
  VAR_INPUT
    sSide : STRING;
  END_VAR
                          METH_IsValidSorterSide := sSide = 'DX' OR sSide = 'SX';
                        
END_METHOD

METHOD METH_SetTESTPhysicalMapping
                          TESTConveyor.aLocations[1].iBufferIndex := 0; // shall be hard-coded depending on the physical implementation
TESTConveyor.aLocations[2].iBufferIndex := 1; // shall be hard-coded depending on the physical implementation
TESTConveyor.aLocations[3].iBufferIndex := 2;
TESTConveyor.aLocations[4].iBufferIndex := 3;

(**)
TESTConveyor.aLocations[5].iBufferIndex := 4; // shall be hard-coded depending on the physical implementation
TESTConveyor.aLocations[6].iBufferIndex := 5; // shall be hard-coded depending on the physical implementation
TESTConveyor.aLocations[7].iBufferIndex := 6;
TESTConveyor.aLocations[8].iBufferIndex := 7;


                        
END_METHOD

METHOD METH_TESTConvertToLocationName
  VAR_INPUT
    Item : items_struct_t;
  END_VAR
                          TESTItem := Item;
xTB_TESTConvert := TRUE;
                        
END_METHOD
END_PROGRAM

PROGRAM prg_hmi_TestSorterSX
  VAR
    asLocationAnim02 : ARRAY[0..19] OF items_struct_t := [(sItemCode := 'BOX_ANIM_02', eLocationType := location_type_enum_t.Conveyor), (sItemCode := 'BOX_ANIM_02', eLocationType := location_type_enum_t.Conveyor, iLocationIndex := 1), (sItemCode := 'BOX_ANIM_02', eLocationType := location_type_enum_t.Conveyor, iLocationIndex := 2), (sItemCode := 'BOX_ANIM_02', eLocationType := location_type_enum_t.Buffer, iLocationIndex := 1), (sItemCode := 'BOX_ANIM_02', eLocationType := location_type_enum_t.Buffer, iLocationIndex := 1, iLocationSubIndex := 1), 2((sItemCode := 'BOX_ANIM_02', eLocationType := location_type_enum_t.Buffer, iLocationIndex := 1, iLocationSubIndex := 2)), (sItemCode := 'BOX_ANIM_02', eLocationType := location_type_enum_t.Buffer, iLocationIndex := 1, iLocationSubIndex := 1), (sItemCode := 'BOX_ANIM_02', eLocationType := location_type_enum_t.Buffer, iLocationIndex := 1), (sItemCode := 'BOX_ANIM_02', eLocationType := location_type_enum_t.Conveyor, iLocationIndex := 2), (sItemCode := 'BOX_ANIM_02', eLocationType := location_type_enum_t.Conveyor, iLocationIndex := 3), (sItemCode := 'BOX_ANIM_02', eLocationType := location_type_enum_t.Conveyor, iLocationIndex := 4), (sItemCode := 'BOX_ANIM_02', eLocationType := location_type_enum_t.Conveyor, iLocationIndex := 5), (sItemCode := 'BOX_ANIM_02', eLocationType := location_type_enum_t.Conveyor, iLocationIndex := 6), (sItemCode := 'BOX_ANIM_02', eLocationType := location_type_enum_t.Conveyor, iLocationIndex := 7), (sItemCode := 'BOX_ANIM_02', eLocationType := location_type_enum_t.Conveyor, iLocationIndex := 8), 4(())];
    xDIS_Animation02 : BOOL;
    iAnimStep02 : INT;
    iAnimInd02 : INT;
    iTMPAnimInd02 : INT;
    tStep02 : TIME := TIME#1s0ms;
    xTB_Animation02 : BOOL;
    sBoxCode02 : STRING := 'BOX_ANIM_02';
    iAnimStep01 : INT;
    xTB_Animation01 : BOOL;
    xReqSent : BOOL;
    asLocationAnim01 : ARRAY[0..9] OF STRING := ['SorterSX-B-BufferFront1', 'SorterSX-B-BufferFront2', 'SorterSX-B-BufferFront3', 'SorterSX-B-Buffer3F'];
    TON_WaitStep : TON;
    tStep01 : TIME := TIME#2s0ms;
    iAnimInd01 : INT;
    iTMPAnimInd01 : INT;
    xAtLeastAvalidLocation : BOOL;
    xDIS_Animation01 : BOOL;
    xNextIndexValid : BOOL;
  END_VAR

                    
ACT_Anim01();

ACT_Anim02();
                  

ACTION ACT_Anim01:
                        xAtLeastAvalidLocation := METH_Anim01_IsValidLocation(iIndex := 0);
xDIS_Animation01 := NOT xAtLeastAvalidLocation;

CASE iAnimStep01 OF
	0:
		IF xTB_Animation01 THEN
			xTB_Animation01 := FALSE;
			xReqSent := FALSE;
			iAnimInd01 := 0;
			TON_WaitStep(IN := FALSE);
			IF METH_Anim01_IsValidLocation(iIndex := iAnimInd01) THEN
				iAnimStep01 := iAnimStep01 + 1;
			ELSE
				iAnimStep01 := 11;
			END_IF
		END_IF
	(*------------------------------------*)
	1: // go to location
		IF NOT xReqSent THEN
			xReqSent := TRUE;
			prg_hmi_Sorter_SX.METH_TESTDrawBox(
				sLocationName := asLocationAnim01[iAnimInd01]
			);
		ELSE
			TON_WaitStep(IN := TRUE, PT := tStep01);
			IF TON_WaitStep.Q THEN
				TON_WaitStep(IN := FALSE);
				xReqSent := FALSE;
				iAnimStep01 := iAnimStep01 + 1;
			END_IF
		END_IF
	(*------------------------------------*)
	2: // get another location
		iTMPAnimInd01 := iAnimInd01 + 1;
		xNextIndexValid := METH_Anim01_IsValidLocation(iIndex := iTMPAnimInd01);
		IF xNextIndexValid THEN
			iAnimInd01 := iTMPAnimInd01;
			iAnimStep01 := 1;
		ELSE
			iAnimStep01 := 10;
		END_IF
	(*------------------------------------*)
	10:
		iAnimStep01 := 0;
	(*------------------------------------*)
	11: // error
		iAnimStep01 := 0;
	(*------------------------------------*)
END_CASE
                      
END_ACTION

ACTION ACT_Anim02:
                        xAtLeastAvalidLocation := METH_Anim02_IsValidLocation(iIndex := 0);
xDIS_Animation02 := NOT xAtLeastAvalidLocation;

CASE iAnimStep02 OF
	0:
		IF xTB_Animation02 THEN
			xTB_Animation02 := FALSE;
			xReqSent := FALSE;
			iAnimInd02 := 0;
			TON_WaitStep(IN := FALSE);
			IF METH_Anim02_IsValidLocation(iIndex := iAnimInd02) THEN
				iAnimStep02 := iAnimStep02 + 1;
			ELSE
				iAnimStep02 := 11;
			END_IF
		END_IF
	(*------------------------------------*)
	1: // go to location
		IF NOT xReqSent THEN
			xReqSent := TRUE;
			prg_hmi_Sorter_SX.METH_TESTConvertToLocationName(
				Item := asLocationAnim02[iAnimInd02]
			);
		ELSE
			TON_WaitStep(IN := TRUE, PT := tStep02);
			IF TON_WaitStep.Q THEN
				TON_WaitStep(IN := FALSE);
				xReqSent := FALSE;
				iAnimStep02 := iAnimStep02 + 1;
			END_IF
		END_IF
	(*------------------------------------*)
	2: // get another location
		iTMPAnimInd02 := iAnimInd02 + 1;
		xNextIndexValid := METH_Anim02_IsValidLocation(iIndex := iTMPAnimInd02);
		IF xNextIndexValid THEN
			iAnimInd02 := iTMPAnimInd02;
			iAnimStep02 := 1;
		ELSE
			iAnimStep02 := 10;
		END_IF
	(*------------------------------------*)
	10:
		iAnimStep02 := 0;
	(*------------------------------------*)
	11: // error
		iAnimStep02 := 0;
	(*------------------------------------*)
END_CASE
                      
END_ACTION

METHOD METH_Anim01_IsIndexValid : BOOL
  VAR_INPUT
    iIndex : INT;
  END_VAR
  VAR
    iMaxIndAnim01 : INT;
  END_VAR
                          iMaxIndAnim01 := TO_INT(XSIZEOF(asLocationAnim01)/XSIZEOF(asLocationAnim01[0])) - 1;

METH_Anim01_IsIndexValid := iIndex >= 0 AND iIndex <= iMaxIndAnim01;

                        
END_METHOD

METHOD METH_Anim01_IsValidLocation : BOOL
  VAR_INPUT
    iIndex : INT;
  END_VAR
  VAR
    xValidIndex : BOOL;
    xRes : BOOL;
    xValidLocation : BOOL;
  END_VAR
                          xValidIndex := METH_Anim01_IsIndexValid(iIndex := iIndex);
IF xValidIndex THEN
	xValidLocation := asLocationAnim01[iIndex] <> '';
	IF xValidLocation THEN
		xRes := TRUE;
	END_IF
END_IF

METH_Anim01_IsValidLocation := xRes;
                        
END_METHOD

METHOD METH_Anim02_IsIndexValid : BOOL
  VAR_INPUT
    iIndex : INT;
  END_VAR
  VAR
    iMaxIndAnim02 : INT;
  END_VAR
                          iMaxIndAnim02 := TO_INT(XSIZEOF(asLocationAnim02)/XSIZEOF(asLocationAnim02[0])) - 1;

METH_Anim02_IsIndexValid := iIndex >= 0 AND iIndex <= iMaxIndAnim02;

                        
END_METHOD

METHOD METH_Anim02_IsValidLocation : BOOL
  VAR_INPUT
    iIndex : INT;
  END_VAR
  VAR
    xValidIndex : BOOL;
    xRes : BOOL;
    xValidLocation : BOOL;
  END_VAR
                          xValidIndex := METH_Anim02_IsIndexValid(iIndex := iIndex);
IF xValidIndex THEN
	xValidLocation := asLocationAnim02[iIndex].eLocationType <> location_type_enum_t.Undefined;
	IF xValidLocation THEN
		xRes := TRUE;
	END_IF
END_IF

METH_Anim02_IsValidLocation := xRes;
                        
END_METHOD
END_PROGRAM

PROGRAM prgDial_ROSPallOpt_A_Left
  VAR
    sToolName : STRING;  (* tool *)
    iIndexToolName : INT;
    sLayerName : STRING;  (* layer *)
    iIndexLayerName : INT;
    sPatternName : STRING;  (* pattern *)
    iIndexPatternName : INT;
    ROSInterface : ros_interface_struct_t;
    PalletizingOptions : PalletizingOptions;
    lrWeight : LREAL := 1.5;
    xIsOccupied : BOOL;
    xDIS_Overwrite : BOOL;
    xDIS_Pattern : BOOL;
    xDIS_Tool : BOOL;
    xDIS_Object : BOOL;
    lrPrevWeight : LREAL;
    sPrevPatternName : STRING;
    sPrevLayerName : STRING;
  END_VAR

                    xDIS_Overwrite := xIsOccupied; // to evaluate

xDIS_Pattern := xDIS_Overwrite;
xDIS_Tool := xDIS_Overwrite;
xDIS_Object := xDIS_Overwrite;
(*---------------------------------------*)
// select info to write
sPatternName := prgObjectCode.asPatternName[iIndexPatternName];
sLayerName := prgObjectCode.asLayerName[iIndexLayerName];
(*---------------------------------------*)
// get current info to show
ROSInterface := prgROS.ROSInterface_01; // EDIT
PalletizingOptions := ROSInterface.Codesys2ROS.Published.lft_palletizing_options; //EDIT
(*---------------------------------------*)
// write variables
IF lrWeight <> lrPrevWeight THEN
	prgROS.METH_SetObjectWeight_Left_01(lrValue := lrWeight);
END_IF
lrPrevWeight := lrWeight;

IF sPatternName <> sPrevPatternName THEN
	prgROS.METH_SetPatternName_Left_01(sValue := sPatternName);
END_IF
sPrevPatternName := sPatternName;

IF sLayerName <> sPrevLayerName THEN
	prgROS.METH_SetTransform_Left_01(sValue := sLayerName);
END_IF
sPrevLayerName := sLayerName;
                  
END_PROGRAM

PROGRAM prgROSInterfaceToLifter01
  VAR
    R_TRIG_Command : Standard.R_TRIG;
    F_TRIG_Command : Standard.F_TRIG;
    xSuccess : BOOL;
    xFailure : BOOL;
    xAborted : BOOL;
    xBusy : BOOL;
    xSimulation : BOOL;
    SIMFeedback : CommonFeedback;
    SIMCommand : CommonCommand;
    diActionID : DINT;
    xCameraDelayCond : BOOL;
    R_TRIG_Success : R_TRIG;
    xExecuteTrigger : BOOL;
    R_TRIG_Abort : R_TRIG;
    REFFeedback : REFERENCE TO CommonFeedback;
    REFCommand : REFERENCE TO CommonCommand;
  END_VAR

                    IF xSimulation THEN
	REFFeedback REF= SIMFeedback;
	REFCommand REF= SIMCommand;
ELSE
	REFFeedback REF= prgROS.ROSInterface_01.Codesys2ROS.Published.lifter_controller_feedback;
	REFCommand REF= prgROS.ROSInterface_01.ROS2Codesys.Subscripted.lifter_controller_command;
END_IF


IF __ISVALIDREF(REFFeedback) AND __ISVALIDREF(REFCommand) THEN
(*======================================*)
	diActionID := REFCommand.id;
	ACT_SerialROSResponse();
// 	CASE diActionID OF
// 		1: // serial action
// 			ACT_SerialROSResponse();
// 		2: // execute and immediate response (at least busy or failed)
// 			ACT_ImmediateROSResponse();
// 		ELSE
// 			ACT_SerialROSResponse();
// 	END_CASE
END_IF

                  

ACTION ACT_SerialROSResponse:
                        // catch triggers of ROS Command

R_TRIG_Command(CLK := REFCommand.execute);
IF R_TRIG_Command.Q THEN
	METH_ClearFeedback();
	prgLifter01.METH_SetAction(diAction := TO_UINT(REFCommand.id));
	prgLifter01.METH_DoNewCycle();
END_IF

R_TRIG_Abort(CLK := REFCommand.abort);
IF R_TRIG_Abort.Q THEN
	prgLifter01.METH_AbortCycle();
END_IF

IF REFCommand.execute THEN
	IF xSuccess THEN
		xSuccess := FALSE;
		REFFeedback.done := TRUE;
		REFFeedback.error := FALSE;
		REFFeedback.aborted := FALSE;
		REFFeedback.error_id := prgLifter01.METH_GetLastErrorID();
	ELSIF xFailure THEN
		xFailure := FALSE;
		REFFeedback.done := FALSE;
		REFFeedback.error := TRUE;
		REFFeedback.aborted := FALSE;
		REFFeedback.error_id := prgLifter01.METH_GetLastErrorID();
	ELSIF xAborted THEN
		xAborted := FALSE;
		REFFeedback.done := FALSE;
		REFFeedback.error := FALSE;
		REFFeedback.aborted := TRUE;
		REFFeedback.error_id := prgLifter01.METH_GetLastErrorID();
	ELSE
		REFFeedback.busy := prgLifter01.METH_IsOccupied();
	END_IF
ELSE
	METH_ClearFeedback();
END_IF
                      
END_ACTION

ACTION ACT_ImmediateROSResponse:
                        // catch triggers of ROS Command

xExecuteTrigger := REFCommand.execute AND GVL.g_xRUNNING;
R_TRIG_Command(CLK := xExecuteTrigger);
IF R_TRIG_Command.Q THEN
	METH_ClearFeedback();
	prgFeeding_B.METH_DoNewCycle();
END_IF

IF xExecuteTrigger THEN
	IF xSuccess OR xBusy THEN // immediate response as soon as busy
		xSuccess := FALSE;
		REFFeedback.done := TRUE;
		REFFeedback.error := FALSE;
		REFFeedback.aborted := FALSE;
	ELSIF xFailure THEN
		xFailure := FALSE;
		REFFeedback.done := FALSE;
		REFFeedback.error := TRUE;
		REFFeedback.aborted := FALSE;
	ELSIF xAborted THEN
		xAborted := FALSE;
		REFFeedback.done := FALSE;
		REFFeedback.error := FALSE;
		REFFeedback.aborted := TRUE;
	ELSE
		REFFeedback.busy := prgFeeding_B.METH_IsOccupied();
	END_IF
ELSE
	METH_ClearFeedback();
END_IF
                      
END_ACTION

METHOD METH_SetSuccess
                          xSuccess := TRUE;
                        
END_METHOD

METHOD METH_SetFailure
                          xFailure := TRUE;
                        
END_METHOD

METHOD METH_SetAborted
                          xAborted := TRUE;
                        
END_METHOD

METHOD METH_SetBusyValue
  VAR_INPUT
    xValue : BOOL;
  END_VAR
                          xBusy := xValue;
                        
END_METHOD

METHOD METH_ClearFeedback
                          IF __ISVALIDREF(REFFeedback) THEN
	SysMemSet(pDest := ADR(REFFeedback), udiCount := XSIZEOF(REFFeedback), udiValue := 0);
END_IF

xSuccess := FALSE;
xFailure := FALSE;
xAborted := FALSE;
xBusy :=  FALSE;
                        
END_METHOD
END_PROGRAM

PROGRAM prgLifter01
  VAR
    xSimulation : BOOL := TRUE;
    CTRL_Axis : SysDesignBasic.SysD_basic_ctrl_abrt_struct_t;
    R_TRIG_Execute : STandard.R_TRIG;
    F_TRIG_Execute : STandard.F_TRIG;
    xSimTimeCond : BOOL;
    tSim : TIME := TIME#3s0ms;
    TON_Sim : TON;
    diActionID : DINT;
    diLastErrorID : DINT;
    R_TRIG_Abort : R_TRIG;
    F_TRIG_Abort : R_TRIG;
    xAbortNow : BOOL;
  END_VAR

                    IF xSimulation THEN
	ACT_Simulation();
ELSE
	//
END_IF
                  

ACTION ACT_Simulation:
                        R_TRIG_Execute(CLK := CTRL_Axis.xExecute);
F_TRIG_Execute(CLK := CTRL_Axis.xExecute);

R_TRIG_Abort(CLK := xSimTimeCond AND CTRL_Axis.xAbort);
F_TRIG_Abort(CLK := CTRL_Axis.xAbort);

IF R_TRIG_Execute.Q THEN
	xSimTimeCond := TRUE;
END_IF
IF R_TRIG_Abort.Q THEN
	xAbortNow := TRUE;
END_IF
TON_Sim(IN := xSimTimeCond, PT := tSim);
IF TON_Sim.Q THEN
	TON_Sim(IN := FALSE);
	xSimTimeCond := FALSE;
	CASE diActionID OF
		0, 1, 2:
			prgROSInterfaceToLifter01.METH_SetSuccess();
			diLastErrorID := 0;
		ELSE
			prgROSInterfaceToLifter01.METH_SetFailure();
			diLastErrorID := 1;
	END_CASE
	CTRL_Axis.xExecute := FALSE;
ELSIF xAbortNow THEN
	xAbortNow := FALSE;
	xSimTimeCond := FALSE;
	prgROSInterfaceToLifter01.METH_SetAborted();
	diLastErrorID := -1;
	CTRL_Axis.xExecute := FALSE;
END_IF
                      
END_ACTION

METHOD METH_IsOccupied : BOOL
                          METH_IsOccupied := CTRL_Axis.xExecute;
                        
END_METHOD

METHOD METH_DoNewCycle : BOOL
                          CTRL_Axis.xExecute := TRUE;
                        
END_METHOD

METHOD METH_SetAction : BOOL
  VAR_INPUT
    diAction : DINT;
  END_VAR
                          diActionID := diAction;
                        
END_METHOD

METHOD METH_GetLastErrorID : DINT
                          METH_GetLastErrorID := diLastErrorID;
                        
END_METHOD

METHOD METH_AbortCycle : BOOL
                          CTRL_Axis.xAbort := TRUE;
                        
END_METHOD
END_PROGRAM

CONFIGURATION Device
  RESOURCE Application ON PLC
    {attribute 'qualified_only'}
    VAR_GLOBAL  (* GVL *)
      g_LightTower : light_tower_struct_t;
      sState : STRING(255) := 'CubeOS';
      sBanner : STRING(255) := 'SysDesign';
      g_xPLAY : BOOL;
      g_xRUNNING : BOOL;
      g_xPAUSE : BOOL;
      g_xRESET : BOOL;
      g_xRESETTING : BOOL;
      g_xSTOP : BOOL;
      g_xRobotError : BOOL;
      g_xPieceError : BOOL;
      g_axVISION_ERROR : ARRAY[0..1] OF BOOL;
      g_xRebootApplication : BOOL;
      g_aMarkerEulPoses : ARRAY[0..1] OF ROS_pose_eu_struct_t;  (* g_ROSInterface_01 : ros_interface_struct_t_OLD; g_ROSInterface_02 : ros_interface_struct_t_OLD; *)
      g_xSafetyOK : BOOL := TRUE;
      g_xSafeguardOK : BOOL := TRUE;
      g_xNODES_START : BOOL;
      g_xNODES_STOP : BOOL;
      g_xShutdownMiniPC : BOOL;
      g_xRebootMiniPC : BOOL;
      g_xListDockers : BOOL;
      g_xLocalTestMachine : BOOL;
      g_xDoosanButton : BOOL;
      g_xDoosanMayBeOff : BOOL;
      g_xDoosanButton_2 : BOOL;
      g_xDoosanMayBeOff_2 : BOOL;
    END_VAR
    {attribute 'qualified_only'}
    VAR_GLOBAL  (* GVL_Applica *)
      g_MachineMESInterface : full_machine_struct_t;
      g_SessionCounters : counters_struct_t;
      g_iDepth : INT := 20;
    END_VAR
    {attribute 'qualified_only'}
    {attribute 'checksumnoinit_override' := '268297182'}
    {attribute 'init_related_code' := 'dd094e88-8960-439b-9848-851b40b15be6'}
    VAR_GLOBAL RETAIN PERSISTENT  (* PersVars *)
      {attribute 'order_in_persistent_editor' := '0'}
      g_OverallCounters : counters_struct_t;
      {attribute 'order_in_persistent_editor' := '1'}
      g_uiCurrentPalletConfig : UINT;
    END_VAR
    {attribute 'qualified_only'}
    VAR_GLOBAL  (* GVL_HMI *)
      xPlay : BOOL;  (* - *)
      xPause : BOOL;
      xReload : BOOL;
      xStop : BOOL;
      xAutoManu : BOOL;
      i_SpeedPerc : INT;
      xLogin : BOOL;  (* - *)
      xLogOut : BOOL;
      xTowerLight_Red : BOOL;  (* - *)
      xTowerLight_Yellow : BOOL;
      xTowerLight_Green : BOOL;
      DisableReboot : BOOL;  (* - xEmergencyMachine:BOOL; *)
      g_xIsStoppedByUser : BOOL;  (* 08/11/2022 *)
      gc_ClientVisu : INT := 100;
    END_VAR
    {attribute 'qualified_only'}
    VAR_GLOBAL CONSTANT  (* GVL_ProcessCode *)
      gc_diProcessUnknown : DINT := 0;
      gc_diPICK_RUNNING : DINT := 20;
      gc_diPICK_FAILED : DINT := -20;
      gc_diPLACE_RUNNING : DINT := 30;
      gc_diPLACE_FAILED : DINT := -30;
      gc_diFINISHED : DINT := 100;
    END_VAR
    {attribute 'qualified_only'}
    VAR_GLOBAL CONSTANT  (* GVL_Constants *)
      gc_dwRed : DWORD := 16#FFFF0000;
      gc_dwGreen : DWORD := 16#FF99FFCC;
      gc_dwBlue : DWORD := 16#FF0000FF;
      gc_dwWhite : DWORD := 16#FFFFFFFF;
      gc_dwYellow : DWORD := 16#FFEEBD28;
      gc_sZeroTimestamp : STRING := 'CONCAT(DT_TO_STRING(ANY_TO_DT(0)), '.000')';
      gc_uiPalletConfigIndex_01 : UINT := 0;
      gc_uiPalletConfigIndex_02 : UINT := 1;
      gc_sTESTDatabaseIP : STRING := '192.168.1.182';
      gc_sTESTDatabaseName : STRING := 'DB_23SH01';
    END_VAR
    {attribute 'qualified_only'}
    VAR_GLOBAL  (* IO_Variables *)
      g_Doosan_EIP : doosan_t;
      g_udiRobotState : UDINT;
      g_Doosan_EIP_2 : doosan_t;
      g_udiRobotState_2 : UDINT;
    END_VAR
    TASK MainTask(INTERVAL := T#100ms, PRIORITY := 31);
    TASK VISU_TASK(INTERVAL := T#100ms, PRIORITY := 31);
    TASK Task_HMI(INTERVAL := T#100ms, PRIORITY := 31);
    TASK ENIPScannerIOTask(INTERVAL := T#10ms, PRIORITY := 0);
    TASK ENIPScannerServiceTask(INTERVAL := T#20ms, PRIORITY := 30);
    TASK TaskFast(INTERVAL := T#20ms, PRIORITY := 31);
    TASK TaskDB(INTERVAL := T#20ms, PRIORITY := 15);
    PROGRAM prgMain WITH MainTask : prgMain;
    PROGRAM prgROS WITH MainTask : prgROS;
    PROGRAM prgApplica WITH MainTask : prgApplica;
    PROGRAM prgLight WITH MainTask : prgLight;
    PROGRAM Reboot_Application WITH MainTask : Reboot_Application;
    PROGRAM prgLinuxCommand WITH MainTask : prgLinuxCommand;
    PROGRAM prgObjectCode WITH MainTask : prgObjectCode;
    PROGRAM prgOPCUAIncas WITH MainTask : prgOPCUAIncas;
    PROGRAM prgInboundSync WITH MainTask : prgInboundSync;
    PROGRAM prgLifter01 WITH MainTask : prgLifter01;
    PROGRAM prgROSInterfaceToLifter01 WITH MainTask : prgROSInterfaceToLifter01;
    PROGRAM VisuElems.Visu_Prg WITH VISU_TASK : VisuElems.Visu_Prg;
    PROGRAM prg_HMI_MainFrame WITH Task_HMI : prg_HMI_MainFrame;
    PROGRAM prg_Hmi_FrameRobotMenu WITH Task_HMI : prg_Hmi_FrameRobotMenu;
    PROGRAM prg_Hmi_FrameMiniPCMenu WITH Task_HMI : prg_Hmi_FrameMiniPCMenu;
    PROGRAM prg_HMI_MiniPCMenu WITH Task_HMI : prg_HMI_MiniPCMenu;
    PROGRAM prg_Hmi_ManagerMiniPC WITH Task_HMI : prg_Hmi_ManagerMiniPC;
    PROGRAM prg_Hmi_Home WITH Task_HMI : prg_Hmi_Home;
    PROGRAM prg_Hmi_Application WITH Task_HMI : prg_Hmi_Application;
    PROGRAM prg_Hmi_RobotMenu WITH Task_HMI : prg_Hmi_RobotMenu;
    PROGRAM prg_Hmi_InterfaceSetting WITH Task_HMI : prg_Hmi_InterfaceSetting;
    PROGRAM prg_Hmi_RobotControl WITH Task_HMI : prg_Hmi_RobotControl;
    PROGRAM prg_Hmi_RobotControl2 WITH Task_HMI : prg_Hmi_RobotControl2;
    PROGRAM prg_Hmi_AskedPose WITH Task_HMI : prg_Hmi_AskedPose;
    PROGRAM prg_Hmi_PalletConfig WITH Task_HMI : prg_Hmi_PalletConfig;
    PROGRAM PLC_PRG WITH Task_HMI : PLC_PRG;
    PROGRAM prg_Hmi_ZoneTractor WITH Task_HMI : prg_Hmi_ZoneTractor;
    PROGRAM prg_Hmi_ObjectCode WITH Task_HMI : prg_Hmi_ObjectCode;
    PROGRAM prg_Hmi_OPCUATests WITH Task_HMI : prg_Hmi_OPCUATests;
    PROGRAM prgDial_ROSInfo_A WITH Task_HMI : prgDial_ROSInfo_A;
    PROGRAM prgDial_ROSInfo_B WITH Task_HMI : prgDial_ROSInfo_B;
    PROGRAM prg_Hmi_RobotSelection WITH Task_HMI : prg_Hmi_RobotSelection;
    PROGRAM prg_hmi_Synoptic WITH Task_HMI : prg_hmi_Synoptic;
    PROGRAM prg_hmi_Sorter_SX WITH Task_HMI : prg_hmi_Sorter_SX;
    PROGRAM prg_hmi_TestSorterSX WITH Task_HMI : prg_hmi_TestSorterSX;
    PROGRAM prgDial_ROSPallOpt_A_Left WITH Task_HMI : prgDial_ROSPallOpt_A_Left;
    PROGRAM EtherNet_IP_Scanner.IOCycle WITH ENIPScannerIOTask : EtherNet_IP_Scanner.IOCycle;
    PROGRAM EtherNet_IP_Scanner.ServiceCycle WITH ENIPScannerServiceTask : EtherNet_IP_Scanner.ServiceCycle;
    PROGRAM prgEIPMapping WITH TaskFast : prgEIPMapping;
    PROGRAM prgDBExecutor WITH TaskDB : prgDBExecutor;
    PROGRAM prgDBQuerier_SorterSX WITH TaskDB : prgDBQuerier_SorterSX;
    PROGRAM prgDBQuerierLogger WITH TaskDB : prgDBQuerierLogger;
  END_RESOURCE
END_CONFIGURATION

CONFIGURATION Ethernet
END_CONFIGURATION

CONFIGURATION EtherNet_IP_Scanner
END_CONFIGURATION

CONFIGURATION DoosanRobot_EIP_Adapter_Monitoring_GPR
END_CONFIGURATION

CONFIGURATION DoosanRobot_EIP_Adapter_Monitoring_GPR_1
END_CONFIGURATION

CONFIGURATION SoftMotion General Axis Pool
END_CONFIGURATION
